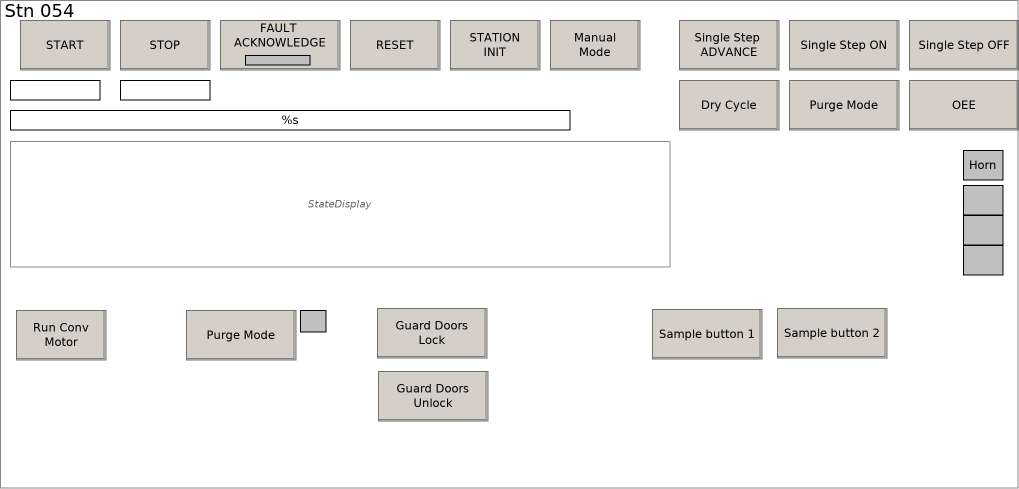
VISUALIZATION Station  // 1019x489
    Button (20,20 90x50), "START"
        tap Global_Variables.gStn054.hiCycleStart
    Button (120,20 90x50), "STOP"
        tap Global_Variables.gStn054.hiCycleStop
    RoundedRectangle (10,80 90x20), colour variable: 16#FF000000 OR (16#FF000000 OR (Stn054_01_HMI.hoStartButtonColor))
    RoundedRectangle (120,80 90x20), colour variable: 16#FF000000 OR (16#FF000000 OR (Stn054_01_HMI.hoStopButtonColor))
    Button (220,20 120x50), "FAULT ACKNOWLEDGE", input disabled if: NOT Stn054_00_ModeControl.SeparateAckAndReset
        tap Global_Variables.gStn054.hiFaultAck
    Button (350,20 90x50), "RESET"
        tap Global_Variables.gStn054.hiFaultReset
    Button (450,20 90x50), "STATION INIT"
        tap Global_Variables.gStn054.hiStationReset
    RoundedRectangle (10,110 560x20), "%s", text variable: gStn054.OperatorMessage.Text, colour variable: 16#FF000000 OR (16#FF000000 OR (Global_Variables.gStn100.OperatorMessage.Color))
    Button (789,20 110x50), "Single Step ON"
        tap Global_Variables.gStn054.hiSingleStepON
    Button (909,20 110x50), "Single Step OFF"
        tap Global_Variables.gStn054.hiSingleStepOff
    Button (679,20 100x50), "Single Step ADVANCE"
        tap Global_Variables.gStn054.hiSingleStepAdvance
    Button (550,20 90x50), "Manual Mode"
        tap Global_Variables.gStn054.hiManualMode
    Button (679,80 100x50), "Dry Cycle", pressed state: Stn054_00_ModeControl.hiStationDryCycleEnable
        toggle Stn054_00_ModeControl.hiStationDryCycleEnable
    Button (789,80 110x50), "Purge Mode", pressed state: Stn054_00_ModeControl.hiStationPurgeModeEnable
        toggle Stn054_00_ModeControl.hiStationPurgeModeEnable
    Button (909,80 110x50), "OEE"
        OnMouseUp: change screen: OEE
    RoundedRectangle (245,55 65x10), colour toggle: NOT Stn054_00_ModeControl.SeparateAckAndReset
    Rectangle (963,185 40x30), colour toggle: Stn054_00_ModeControl.oStackLightRed
    Rectangle (963,215 40x30), colour toggle: Stn054_00_ModeControl.oStackLightAmber
    Rectangle (963,245 40x30), colour toggle: Stn054_00_ModeControl.oStackLightGreen
    Rectangle (963,150 40x30), "Horn", colour toggle: (Stn054_00_ModeControl.oStackLightHorn) <> 0
    Rectangle (636,362 81x30)
    Rectangle (632,459 81x30)
    Frame (10,141 660x126)
        shows StateDisplay()
    Button (16,310 90x50), "Run Conv Motor"
    Label (6,2 67x18), "Stn 054"
    Button (377,308 110x50), "Guard Doors Lock"
        tap Stn054_00_ModeControl.hiGuardDoorsLock
    Button (378,371 110x50), "Guard Doors Unlock"
        tap Stn054_00_ModeControl.hiGuardDoorsUnlock
    Button (652,309 110x50), "Sample button 1"
        tap Stn100_60_TrayUnload.fbTrayCart.hiCartUndockReq
    Button (777,308 110x50), "Sample button 2"
        tap Stn100_20_TrayLoad.fbTrayCart.hiCartUndockReq
    Button (186,310 110x50), "Purge Mode"
        tap Stn100_10_Main.hiPurgeModeToggle
    Rectangle (300,310 26x22), colour toggle: Stn100_10_Main.PurgeModeActive
END_VISUALIZATION

(* stored: Version 1.1.0.1, ProductVersion 3.1.4024.6
   Visu Station: Id {52e31f76-1902-48fd-a5e0-a0a109f1fb31} *)
